FUNCTION_BLOCK FB_HRU EXTENDS FB_CtrlBase
VAR_INPUT
	/// Sensor input
	In_bolHangerDetected: BOOL;
END_VAR
VAR_OUTPUT
	/// Pneumatic cylinder
	Out_bolRotate: BOOL;
	/// Pneumatic cylinder
	Out_bolEject: BOOL;
END_VAR
VAR
	/// Specific interface struct for public access
	SIf: T_Ctrl_SIf_HRU;
	/// Function specific variables
	stSubState: T_Ctrl_Class_StateMachine;
END_VAR
VAR CONSTANT
	///sub States for RELEASE Function
	cSTA_SUB_WAIT_FOR_JOB: INT := 501;
	cSTA_SUB_WAIT_WITH_HANGER: INT := 510;
	cSTA_SUB_ROTATE: INT := 520;
	cSTA_SUB_EJECT: INT := 530;
	cSTA_SUB_RETRACT: INT := 540;
	cSTA_SUB_DONE: INT := 550;
	cSTA_SUB_ERROR: INT := 590;
END_VAR

(*__________________________________________________________________________________________________
¦	
¦	Vistaprint Schweiz GmbH
¦	CH - 8401 Winterthur
¦
¦	www.vistaprint.ch - info@vistaprint.ch
¦___________________________________________________________________________________________________

Function desription:
Hanger rotation unit implementation. 


History:
Version		Date			Author		Comment
---------------------------------------------------------------------------------------------------
0.00.1		25.04.2013		AVME/KVO	Start history
0.00.2		18.09.2013		AVME/MRU	Copied from CYL and renamed to HRU

___________________________________________________________________________________________________*)


IF (me.bolActivate) THEN // cyclic call enabled
	IF (CIf.Info.bolInitDone=FALSE) THEN // first cycle -> init
		CtrlInit();
		CIf.Info.bolInitDone := TRUE;
	ELSE
		CycleStartDuty();
	
		Always();
		
		StateMachine();
		
		CycleEndDuty();
	END_IF
END_IF;

METHOD PROTECTED getCmdState : STRING
VAR_INPUT
	intCmdState: INT;
	bolState: BOOL;
END_VAR
getCmdState := SUPER^.getCmdState(intCmdState:=intCmdState,bolState:=bolState); // get global/base defined cmds/states
IF (getCmdState='') THEN // global not defined get local
	// get string cmd/state string information in runtime
	IF (bolState=FALSE) THEN
		// cmd's
		CASE intCmdState OF
			cCMD_RETRACT: 
				getCmdState := 'cCMD_RETRACT';
			cCMD_EJECT: 
				getCmdState := 'cCMD_EJECT';
			cCMD_ROTATE: 
				getCmdState := 'cCMD_ROTATE';
			cCMD_RUN: 
				getCmdState := 'cCMD_RUN';
		END_CASE;
	ELSE
	
	// states
		CASE intCmdState OF
			cSTA_RETRACTBusy: 
				getCmdState := 'cSTA_RETRACTBusy';
			cSTA_RETRACT: 
				getCmdState := 'cSTA_RETRACT';
			cSTA_EJECTBusy: 
				getCmdState := 'cSTA_EJECTBusy';
			cSTA_EJECT: 
				getCmdState := 'cSTA_EJECT';
			cSTA_ROTATEBusy: 
				getCmdState := 'cSTA_ROTATEBusy';
			cSTA_ROTATE: 
				getCmdState := 'cSTA_ROTATE';
			cSTA_RUNBusy: 
				getCmdState := 'cSTA_RUNBusy';
			cSTA_RUN: 
				getCmdState := 'cSTA_RUN';
				
			// SUB states
			cSTA_SUB_WAIT_FOR_JOB:
				getCmdState := 'cSTA_SUB_WAIT_FOR_JOB';
			cSTA_SUB_WAIT_WITH_HANGER:
				getCmdState := 'cSTA_SUB_WAIT_WITH_HANGER';
			cSTA_SUB_ROTATE:
				getCmdState := 'cSTA_SUB_ROTATE';
			cSTA_SUB_EJECT:
				getCmdState := 'cSTA_SUB_EJECT';
			cSTA_SUB_RETRACT:
				getCmdState := 'cSTA_SUB_RETRACT';
			cSTA_SUB_DONE:
				getCmdState := 'cSTA_SUB_DONE';
			cSTA_SUB_ERROR:
				getCmdState := 'cSTA_SUB_ERROR';

		END_CASE;
	END_IF
END_IF
END_METHOD

METHOD FB_init : BOOL
VAR_INPUT
	///if TRUE, the retain variables are initialized (warm start / cold start)
	bInitRetains: BOOL;
	///if TRUE, the instance afterwards gets moved into the copy code (online change)
	bInCopyCode: BOOL;
END_VAR
VAR
	ii: UINT;
END_VAR
//------------------------------------------------------------------------------------------------------------------------
// to manually change in new FUB implementation!!!
// define valid commands for this controller
FOR ii:= 0 TO (SIZEOF(CIf.Job.aCmdList)/SIZEOF(CIf.Job.aCmdList[0])-1) BY 1 DO
	IF (CIf.Job.aCmdList[ii].intCmd=cCMD_INITIALIZED) THEN
		// found first empty array element
		EXIT;
	END_IF
END_FOR
CIf.Job.aCmdList[ii].intCmd := cCMD_STOP;
CIf.Job.aCmdList[ii].strName := 'Stop'; 
CIf.Job.aCmdList[ii].bolAvailable := TRUE;
ii := ii +1;
CIf.Job.aCmdList[ii].intCmd := cCMD_RETRACT;
CIf.Job.aCmdList[ii].strName := 'Retract';
CIf.Job.aCmdList[ii].bolAvailable := TRUE;
ii := ii +1;
CIf.Job.aCmdList[ii].intCmd := cCMD_EJECT; // for test simulation single answer
CIf.Job.aCmdList[ii].strName := 'EJECT';
CIf.Job.aCmdList[ii].bolAvailable := TRUE;
ii := ii +1;
CIf.Job.aCmdList[ii].intCmd := cCMD_ROTATE; //  MRU 18.09.2013: New command rotate
CIf.Job.aCmdList[ii].strName := 'Rotate'; 
CIf.Job.aCmdList[ii].bolAvailable := TRUE;
ii := ii +1;
CIf.Job.aCmdList[ii].intCmd := cCMD_RUN; // for test simulation single answer
CIf.Job.aCmdList[ii].strName := 'RUN';
CIf.Job.aCmdList[ii].bolAvailable := TRUE;

// set name of class/typ
CIf.Info.strType := 'FB_HRU';

// set alarm class
SIf.Alm[1].eAlmClass := E_AlmClass.TSTOP;
SIf.Alm[1].strText := 'sensor hangerDetected always on'; 
SIf.Alm[2].eAlmClass := E_AlmClass.TSTOP;
SIf.Alm[2].strText := 'sensor hangerDetected always on';
SIf.Alm[3].eAlmClass := E_AlmClass.TSTOP;
SIf.Alm[3].strText := 'sensor hangerDetected always on';
SIf.Alm[4].eAlmClass := E_AlmClass.TSTOP;
SIf.Alm[4].strText := 'Expected Hanger not in Rotation Unit';

//*******************************************************************************
// initial values
//*******************************************************************************

// software configuration
CIf.SwCfg.bolExist := TRUE;
CIf.SwCfg.bolSimulation := FALSE;

// parmeter
SIf.Par.udiEjectTime_ms := 1000;			// No sensor, work with time
SIf.Par.udiRetractTime_ms := 1000;			// No sensor, work with time
SIf.Par.udiRotateTime_ms := 2000;			// No sensor, work with time
SIf.Par.udiWaitForRotate_ms := 4000;		// No sensor, work with time
SIf.Par.udiSimNextHangerTime_ms := 5000;	// For simulation
SIf.Par.udiTimeOutHRU_Hanger_ms := 10000;	// Time out no hanger in rotation unit
END_METHOD

METHOD PROTECTED sta_RETRACTBusy : BOOL
// state implemetation
//--------------------------------------------------------------------------------------
// Entry action
	IF (me.StateMachine.intState<>me.StateMachine.intStateLastCycle) THEN
		me.StateMachine.intStateLastCycle := me.StateMachine.intState;
		
		SIf.Out.bolEject.intern := FALSE;	// Eject Cylinder Valve
		
	END_IF


//--------------------------------------------------------------------------------------
// Cyclic action
	IF (me.StateMachine.intState=me.StateMachine.intStateLastCycle) THEN

		// Simulation
		IF (CIf.SwCfg.bolSimulation) THEN
			;
		END_IF
		
		// State Change Condition
		IF (me.StateMachine.udiTimeInState_ms>SIf.Par.udiRetractTime_ms) THEN
			// Cylinder retracted
			me.StateMachine.intStateNext := cSTA_RETRACT;	
			// timeout extend cylinder 		// Used, if a sensor exist
			// pfbAlarmCtrl^.setAlarm(CIf.Info.intCtrlId,4,0,ADR(SIf.Alm),E_AlmState.RST,CIf.Job.eMe_ActivAlmClass);
			// ELSIF (SIf.In.bolHangerDetected.intern) AND(SIf.In.bolHangerDetected.intern=FALSE) THEN		// Used, if a sensor exist
			// 	me.StateMachine.intStateNext := cSTA_RETRACT;
		ELSIF(me.intCmd=cCMD_STOP) THEN
			me.StateMachine.intStateNext := cSTA_STOPBusy;
		ELSIF(me.intCmd=cCMD_EJECT) THEN
			me.StateMachine.intStateNext := cSTA_EJECTBusy;
		END_IF
	END_IF




//--------------------------------------------------------------------------------------
// Exit action
	IF (me.StateMachine.intState<>me.StateMachine.intStateNext) THEN
		//SIf.Cur.udiMoveTimeRetract := me.StateMachine.udiTimeInState_ms;
		;
	END_IF
END_METHOD

METHOD PROTECTED sta_EJECT : BOOL
// state implemetation
//--------------------------------------------------------------------------------------
// Entry action
	IF (me.StateMachine.intState<>me.StateMachine.intStateLastCycle) THEN
		me.StateMachine.intStateLastCycle := me.StateMachine.intState;

	END_IF


//--------------------------------------------------------------------------------------
// Cyclic action
	IF (me.StateMachine.intState=me.StateMachine.intStateLastCycle) THEN

		// Simulation
		IF (CIf.SwCfg.bolSimulation) THEN
			;
		END_IF
		
		// State Change Condition
		IF (SIf.In.bolHangerDetected.intern) THEN
			// sensor retract always on
			pfbAlarmCtrl^.setAlarm(CIf.Info.intCtrlId,2,0,ADR(SIf.Alm),E_AlmState.RST,CIf.Job.eMe_ActivAlmClass);
			me.StateMachine.intStateNext :=  cSTA_ERROR;
		ELSIF(me.intCmd=cCMD_STOP) THEN
			me.StateMachine.intStateNext := cSTA_STOPBusy;
		ELSIF(me.intCmd=HRU_CmdState.cCMD_RETRACT) THEN
			me.StateMachine.intStateNext := cSTA_RETRACTBusy;
		ELSIF(me.intCmd=HRU_CmdState.cCMD_ROTATE) THEN
			me.StateMachine.intStateNext := cSTA_ROTATEBusy;		
		ELSIF(me.intCmd=cCMD_RUN) THEN
			me.StateMachine.intStateNext := cSTA_RUNBusy;
		END_IF
	END_IF




//--------------------------------------------------------------------------------------
// Exit action
	IF (me.StateMachine.intState<>me.StateMachine.intStateNext) THEN
		;
	END_IF
END_METHOD

METHOD PROTECTED sta_STOP : BOOL
// state implemetation
//--------------------------------------------------------------------------------------
// Entry action
	IF (me.StateMachine.intState<>me.StateMachine.intStateLastCycle) THEN
		me.StateMachine.intStateLastCycle := me.StateMachine.intState;
		
	END_IF


//--------------------------------------------------------------------------------------
// Cyclic action
	IF (me.StateMachine.intState=me.StateMachine.intStateLastCycle) THEN
		
		;
		
		
		// State Change Condition
		IF (me.intCmd=cCMD_OFF) THEN
			// sensor retract always on cylinder
			me.StateMachine.intStateNext :=  cSTA_OFFBusy;
		ELSIF (me.intCmd=cCMD_EJECT) THEN 
			me.StateMachine.intStateNext := cSTA_EJECTBusy;
		ELSIF(me.intCmd=cCMD_RETRACT) THEN
			me.StateMachine.intStateNext := cSTA_RETRACTBusy;
		ELSIF(me.intCmd=cCMD_ROTATE) THEN
			me.StateMachine.intStateNext := cSTA_ROTATEBusy;
		ELSIF (me.intCmd=cCMD_RUN) THEN
			me.StateMachine.intStateNext := cSTA_RUNBusy;
		END_IF
	END_IF




//--------------------------------------------------------------------------------------
// Exit action
	IF (me.StateMachine.intState<>me.StateMachine.intStateNext) THEN
		;
	END_IF
END_METHOD

METHOD PROTECTED sta_RETRACT : BOOL
// state implemetation
//--------------------------------------------------------------------------------------
// Entry action
	IF (me.StateMachine.intState<>me.StateMachine.intStateLastCycle) THEN
		me.StateMachine.intStateLastCycle := me.StateMachine.intState;

	END_IF


//--------------------------------------------------------------------------------------
// Cyclic action
	IF (me.StateMachine.intState=me.StateMachine.intStateLastCycle) THEN

		// Simulation
		IF (CIf.SwCfg.bolSimulation) THEN
			;
		END_IF
		
		// State Change Condition
		IF(me.intCmd=cCMD_STOP) THEN
			me.StateMachine.intStateNext := cSTA_STOPBusy;
		ELSIF(me.intCmd=HRU_CmdState.cCMD_EJECT) THEN
			me.StateMachine.intStateNext := cSTA_EJECTBusy;
		ELSIF(me.intCmd=HRU_CmdState.cCMD_ROTATE) THEN
			me.StateMachine.intStateNext := cSTA_ROTATEBusy;
		ELSIF(me.intCmd=cCMD_RUN) THEN
			me.StateMachine.intStateNext := cSTA_RUNBusy;
		END_IF
	END_IF




//--------------------------------------------------------------------------------------
// Exit action
	IF (me.StateMachine.intState<>me.StateMachine.intStateNext) THEN
		;
	END_IF
END_METHOD

METHOD PROTECTED sta_RUNBusy : BOOL
// state implemetation
//--------------------------------------------------------------------------------------
// Entry action
	IF (me.StateMachine.intState<>me.StateMachine.intStateLastCycle) THEN
		me.StateMachine.intStateLastCycle := me.StateMachine.intState;

		me.SubStateMachine.intState := cSTA_SUB_WAIT_FOR_JOB; 		// init sub state machine
		me.SubStateMachine.intStateNext := cSTA_SUB_WAIT_FOR_JOB; 	// init sub state machine
		
		fbSimulationTimer.IN := FALSE;
		fbSimulationTimer.PT := UDINT_TO_TIME(SIf.Par.udiSimNextHangerTime_ms);
		fbSimulationTimer(); // set time/reset timer
		//fbSimulationTimer.IN := TRUE; // start timer
	END_IF


//--------------------------------------------------------------------------------------
// Cyclic action
	IF (me.StateMachine.intState=me.StateMachine.intStateLastCycle) THEN

		// Simulation
		IF (CIf.SwCfg.bolSimulation) THEN
			fbSimulationTimer(); // simulation time
		END_IF

		//--------------------------------------------------------------------------------------
		// sub state machine for sequence
		CASE me.SubStateMachine.intState OF
			cSTA_SUB_WAIT_FOR_JOB:
				IF (me.SubStateMachine.intState<>me.SubStateMachine.intStateLastCycle) THEN
					me.SubStateMachine.intStateLastCycle := me.SubStateMachine.intState;
				END_IF
				
				// Simulation
				IF (CIf.SwCfg.bolSimulation AND NOT SIf.In.bolHangerDetected.intern) THEN
					fbSimulationTimer.IN := TRUE; // start timer
				END_IF
				IF (fbSimulationTimer.Q) THEN
					SIf.In.bolHangerDetected.intern := TRUE; 	// Hanger in HRU
					fbSimulationTimer.IN := FALSE; 				// Stop timer
				END_IF
				
				// State Change Condition
				// Check error if possible
				IF (SIf.In.bolHangerDetected.intern) THEN
					me.SubStateMachine.intStateNext := cSTA_SUB_WAIT_WITH_HANGER;
				END_IF
				
				// Time out expected hanger is not arrived
				IF (me.SubStateMachine.udiTimeInState_ms > SIf.Par.udiTimeOutHRU_Hanger_ms) THEN	// Hanger Rotation Unit time out waiting
					pfbAlarmCtrl^.setAlarm(CIf.Info.intCtrlId,4,0,ADR(SIf.Alm),E_AlmState.RST,CIf.Job.eMe_ActivAlmClass);
					me.SubStateMachine.intStateNext := cSTA_SUB_ERROR;
				END_IF
		//--------------------------------------------------------------------------------------
			cSTA_SUB_WAIT_WITH_HANGER:
				IF (me.SubStateMachine.intState<>me.SubStateMachine.intStateLastCycle) THEN
					me.SubStateMachine.intStateLastCycle := me.SubStateMachine.intState;
				END_IF
				
				// State Change Condition
				// Check error if possible
				IF (me.SubStateMachine.udiTimeInState_ms >= SIf.Par.udiWaitForRotate_ms) THEN
					me.SubStateMachine.intStateNext := cSTA_SUB_ROTATE;
				END_IF
		//--------------------------------------------------------------------------------------
			cSTA_SUB_ROTATE:
				IF (me.SubStateMachine.intState<>me.SubStateMachine.intStateLastCycle) THEN
					me.SubStateMachine.intStateLastCycle := me.SubStateMachine.intState;
					SIf.Out.bolRotate.intern := NOT SIf.Out.bolRotate.intern;	// Rotate in other direction
				END_IF
				
				
				// State Change Condition
				// Check error if possible
				IF (me.SubStateMachine.udiTimeInState_ms >= SIf.Par.udiRotateTime_ms) THEN
					me.SubStateMachine.intStateNext := cSTA_SUB_EJECT;
				END_IF
		//--------------------------------------------------------------------------------------
			cSTA_SUB_EJECT:
				IF (me.SubStateMachine.intState<>me.SubStateMachine.intStateLastCycle) THEN
					me.SubStateMachine.intStateLastCycle := me.SubStateMachine.intState;
				END_IF
				
				SIf.Out.bolEject.intern := TRUE;	// Eject Cylinder Valve
				
				// Simulation
				IF (CIf.SwCfg.bolSimulation) THEN
					SIf.In.bolHangerDetected.intern := FALSE; // Hanger is leaving the HRU
				END_IF
				
				// State Change Condition
				// Check error if possible
				IF (me.SubStateMachine.udiTimeInState_ms > SIf.Par.udiEjectTime_ms) THEN
					IF (SIf.In.bolHangerDetected.intern) THEN
					// sensor Hanger detected always on
						pfbAlarmCtrl^.setAlarm(CIf.Info.intCtrlId,3,0,ADR(SIf.Alm),E_AlmState.RST,CIf.Job.eMe_ActivAlmClass);
						me.SubStateMachine.intStateNext := cSTA_SUB_ERROR;
					ELSE
						// Hanger ejected
						me.SubStateMachine.intStateNext := cSTA_SUB_RETRACT;
					END_IF
				END_IF
		//--------------------------------------------------------------------------------------
			cSTA_SUB_RETRACT:
				IF (me.SubStateMachine.intState<>me.SubStateMachine.intStateLastCycle) THEN
					me.SubStateMachine.intStateLastCycle := me.SubStateMachine.intState;
				END_IF
				
				SIf.Out.bolEject.intern := FALSE;	// Eject Cylinder Valve

				// State Change Condition
				// Check error if possible
				IF (me.SubStateMachine.udiTimeInState_ms >= SIf.Par.udiRetractTime_ms) THEN
					me.SubStateMachine.intStateNext := cSTA_SUB_DONE;
				END_IF
		//--------------------------------------------------------------------------------------
			cSTA_SUB_DONE:
				//CIf.Job.intACmd:=cSTA_DONE; 	// Not necessary
				;								// do nothing, just for state change
		//--------------------------------------------------------------------------------------
			cSTA_SUB_ERROR:
				IF (me.SubStateMachine.intState<>me.SubStateMachine.intStateLastCycle) THEN
					me.SubStateMachine.intStateLastCycle := me.SubStateMachine.intState;
				END_IF
				
				SIf.Out.bolEject.intern := FALSE;	// Eject Cylinder Valve
				
				// State Change Condition
				// No change, going over an other main state
		//--------------------------------------------------------------------------------------
		END_CASE
		
		// Do in every cycle
		CIf.Job.strSubState := THIS^.getCmdState(intCmdState:=me.SubStateMachine.intState,bolState:=TRUE);
		IF (me.SubStateMachine.intState<>me.SubStateMachine.intStateNext) THEN
			me.SubStateMachine.intState := me.SubStateMachine.intStateNext;  // set next state for next cycle
			me.SubStateMachine.udiTimeInState_ms := 0; // reset timer
			// log state change -> open point
		ELSE
			// increment time in state	
			me.SubStateMachine.udiTimeInState_ms := me.SubStateMachine.udiTimeInState_ms + me.FUBInfo.udiSample_ms;
		END_IF
		
				
		// State Change Condition	
		IF me.SubStateMachine.intState = cSTA_SUB_ERROR THEN
			me.StateMachine.intStateNext :=  cSTA_ERROR;
		ELSIF(me.SubStateMachine.intState = cSTA_SUB_DONE) THEN
			me.StateMachine.intStateNext := cSTA_RUN;
		ELSIF((me.SubStateMachine.intState = cSTA_SUB_WAIT_FOR_JOB) AND(me.intCmd=cCMD_STOP)) THEN
			me.StateMachine.intStateNext := cSTA_STOPBusy;
		//ELSIF((me.SubStateMachine.intState = cSTA_SUB_WAIT_FOR_JOB) AND(me.intCmd=cCMD_OFF)) THEN // Done by BaseCtrl.Always
		//	me.StateMachine.intStateNext := cSTA_OFFBusy;
		END_IF
	END_IF


//--------------------------------------------------------------------------------------
// Exit action
	IF (me.StateMachine.intState<>me.StateMachine.intStateNext) THEN
		;
	END_IF
END_METHOD

METHOD PROTECTED sta_RUN : BOOL
// state implemetation
//--------------------------------------------------------------------------------------
// Entry action
	IF (me.StateMachine.intState<>me.StateMachine.intStateLastCycle) THEN
		me.StateMachine.intStateLastCycle := me.StateMachine.intState;
				
	END_IF


//--------------------------------------------------------------------------------------
// Cyclic action
	IF (me.StateMachine.intState=me.StateMachine.intStateLastCycle) THEN

		// Simulation
		IF (CIf.SwCfg.bolSimulation) THEN
			;
		END_IF
		
		// Cyclicle action
		
		
		// State Change Condition
		IF (TRUE) THEN		// Stop after every cycle -> cSTA_DONE
			me.StateMachine.intStateNext := cSTA_STOPBusy;
		ELSIF (me.intCmd=cCMD_STOP) THEN
			me.StateMachine.intStateNext :=  cSTA_STOPBusy;	
		END_IF
	END_IF


//--------------------------------------------------------------------------------------
// Exit action
	IF (me.StateMachine.intState<>me.StateMachine.intStateNext) THEN
		;
	END_IF
END_METHOD

METHOD getCtrlSIf : POINTER TO T_Ctrl_SIf_HRU
getCtrlSIf := ADR(SIf);
END_METHOD

METHOD PROTECTED sta_ROTATEBusy : BOOL
// state implemetation
//--------------------------------------------------------------------------------------
// Entry action
	IF (me.StateMachine.intState<>me.StateMachine.intStateLastCycle) THEN
		me.StateMachine.intStateLastCycle := me.StateMachine.intState;
		
		SIf.Out.bolRotate.intern := NOT SIf.Out.bolRotate.intern;	// Rotate in other direction
		
	END_IF


//--------------------------------------------------------------------------------------
// Cyclic action
	IF (me.StateMachine.intState=me.StateMachine.intStateLastCycle) THEN

		// Simulation
		IF (CIf.SwCfg.bolSimulation) THEN
			;
		END_IF
		
		// State Change Condition
		IF (me.StateMachine.udiTimeInState_ms>SIf.Par.udiRotateTime_ms) THEN
			me.StateMachine.intStateNext :=  cSTA_ROTATE;
		ELSIF(me.intCmd=cCMD_OFF) THEN
			me.StateMachine.intStateNext := cSTA_OFFBusy;
		ELSIF(me.intCmd=cCMD_STOP) THEN
			me.StateMachine.intStateNext := cSTA_STOPBusy;
		END_IF
	END_IF




//--------------------------------------------------------------------------------------
// Exit action
	IF (me.StateMachine.intState<>me.StateMachine.intStateNext) THEN
		//SIf.Cur.udiMoveTimeRetract := me.StateMachine.udiTimeInState_ms;
		;
	END_IF
END_METHOD

METHOD PROTECTED sta_STOPBusy : BOOL
// state implemetation
//--------------------------------------------------------------------------------------
// Entry action
	IF (me.StateMachine.intState<>me.StateMachine.intStateLastCycle) THEN
		me.StateMachine.intStateLastCycle := me.StateMachine.intState;
		
	END_IF


//--------------------------------------------------------------------------------------
// Cyclic action
	IF (me.StateMachine.intState=me.StateMachine.intStateLastCycle) THEN
		
		// switch off?
		// SIf.Out.bolEject.intern := FALSE;	// Eject Cylinder Valve
		
		// State Change Condition
		IF (FALSE) THEN
			;
		ELSIF (TRUE) THEN
			me.StateMachine.intStateNext := cSTA_STOP;
		END_IF
	END_IF




//--------------------------------------------------------------------------------------
// Exit action
	IF (me.StateMachine.intState<>me.StateMachine.intStateNext) THEN
		;
	END_IF
END_METHOD

METHOD PROTECTED sta_OFF : BOOL
// state implemetation
//--------------------------------------------------------------------------------------
// Entry action
	IF (me.StateMachine.intState<>me.StateMachine.intStateLastCycle) THEN
		me.StateMachine.intStateLastCycle := me.StateMachine.intState;
		
	END_IF


//--------------------------------------------------------------------------------------
// Cyclic action
	IF (me.StateMachine.intState=me.StateMachine.intStateLastCycle) THEN
		
		;
		
		
		// State Change Condition
		IF (me.intCmd=cCMD_STOP) THEN
			me.StateMachine.intStateNext :=  cSTA_STOPBusy;
		ELSIF (me.intCmd=HRU_CmdState.cCMD_EJECT) THEN 
			me.StateMachine.intStateNext := cSTA_EJECTBusy;
		ELSIF(me.intCmd=HRU_CmdState.cCMD_RETRACT) THEN
			me.StateMachine.intStateNext := cSTA_RETRACTBusy;
		ELSIF(me.intCmd=HRU_CmdState.cCMD_ROTATE) THEN
			me.StateMachine.intStateNext := cSTA_ROTATEBusy;
		ELSIF(me.intCmd=cCMD_RUN) THEN
			me.StateMachine.intStateNext := cSTA_RUNBusy;
		END_IF
	END_IF




//--------------------------------------------------------------------------------------
// Exit action
	IF (me.StateMachine.intState<>me.StateMachine.intStateNext) THEN
		;
	END_IF
END_METHOD

METHOD PROTECTED sta_OFFBusy : BOOL
// state implemetation
//--------------------------------------------------------------------------------------
// Entry action
	IF (me.StateMachine.intState<>me.StateMachine.intStateLastCycle) THEN
		me.StateMachine.intStateLastCycle := me.StateMachine.intState;
		
	END_IF


//--------------------------------------------------------------------------------------
// Cyclic action
	IF (me.StateMachine.intState=me.StateMachine.intStateLastCycle) THEN
		
		// switch off?
		// SIf.Out.bolEject.intern := FALSE;	// Eject Cylinder Valve
		
		// State Change Condition
		IF (FALSE) THEN
			;
		ELSIF (TRUE) THEN
			me.StateMachine.intStateNext := cSTA_OFF;
		END_IF
	END_IF




//--------------------------------------------------------------------------------------
// Exit action
	IF (me.StateMachine.intState<>me.StateMachine.intStateNext) THEN
		;
	END_IF
END_METHOD

METHOD PROTECTED IoOutBridge : BOOL
// digitale and analoge inputs read from hardware or forcing
IF (CIf.SwCfg.bolSimulation = FALSE) THEN
	setOutBol(CIf.Job.bolIoForce ,ADR(SIf.Out.bolEject));
	setOutBol(CIf.Job.bolIoForce ,ADR(SIf.Out.bolRotate));
	
	THIS^.Out_bolEject := SIf.Out.bolEject.map;
	THIS^.Out_bolRotate := SIf.Out.bolRotate.map;
END_IF
END_METHOD

METHOD PROTECTED StateMachine : BOOL
SUPER^.StateMachine();

// main statemachine of base controller
CASE me.StateMachine.intState OF
	cSTA_ROTATEBusy: 
        THIS^.sta_ROTATEBusy();
    cSTA_ROTATE: 
        THIS^.sta_ROTATE();
	cSTA_RETRACTBusy: 
        THIS^.sta_RETRACTBusy();
    cSTA_RETRACT: 
        THIS^.sta_RETRACT();
    cSTA_EJECTBusy:				// Eject 
        THIS^.sta_EJECTBusy();
    cSTA_EJECT: 
        THIS^.sta_EJECT();
	cSTA_RUNBusy: 
        THIS^.sta_RUNBusy();	// Auto (Wait - Rotate - Eject - Retract)
    cSTA_RUN: 
        THIS^.sta_RUN();
	cSTA_STOPBusy: 				// Rotate rests in his Position, Ejector in Retract Position
        THIS^.sta_STOPBusy();
    cSTA_STOP: 
        THIS^.sta_STOP();
		
END_CASE;
END_METHOD

METHOD PROTECTED sta_EJECTBusy : BOOL
// state implemetation
//--------------------------------------------------------------------------------------
// Entry action
	IF (me.StateMachine.intState<>me.StateMachine.intStateLastCycle) THEN
		me.StateMachine.intStateLastCycle := me.StateMachine.intState;

	END_IF


//--------------------------------------------------------------------------------------
// Cyclic action
	IF (me.StateMachine.intState=me.StateMachine.intStateLastCycle) THEN

		// Simulation
		IF (CIf.SwCfg.bolSimulation) THEN
			;
		END_IF
		
		//no change action
		SIf.Out.bolEject.intern := TRUE;	// Eject Cylinder Valve
		
		
		// State Change Condition
		IF (me.StateMachine.udiTimeInState_ms>SIf.Par.udiEjectTime_ms) THEN
			IF (SIf.In.bolHangerDetected.intern) THEN
				// sensor Hanger detected always on
				pfbAlarmCtrl^.setAlarm(CIf.Info.intCtrlId,1,0,ADR(SIf.Alm),E_AlmState.RST,CIf.Job.eMe_ActivAlmClass);
				me.StateMachine.intStateNext :=  cSTA_ERROR;
			ELSE
				// Hanger ejected
				me.StateMachine.intStateNext := cSTA_EJECT;	
			END_IF
		ELSIF(me.intCmd=cCMD_STOP) THEN
			me.StateMachine.intStateNext := cSTA_STOPBusy;
		ELSIF(me.intCmd=HRU_CmdState.cCMD_RETRACT) THEN
			me.StateMachine.intStateNext := cSTA_RETRACTBusy;
		END_IF
	END_IF




//--------------------------------------------------------------------------------------
// Exit action
	IF (me.StateMachine.intState<>me.StateMachine.intStateNext) THEN
		;
	END_IF
END_METHOD

METHOD PROTECTED IoInBridge : BOOL
// digitale and analoge inputs read from hardware or forcing
SIf.In.bolHangerDetected .map := THIS^.In_bolHangerDetected;

IF (CIf.SwCfg.bolSimulation = FALSE) THEN
	getInBol(CIf.Job.bolIoForce,ADR(SIf.In.bolHangerDetected));
ELSE
	//simulation of global IO
END_IF
END_METHOD

METHOD PROTECTED Always : BOOL
SUPER^.Always();

IF (me.StateMachine.intState<>cSTA_SINGLE_ANSWER) THEN
	;
END_IF


// Always change actions in Base Library
// ----------------------------------------------------------------------------------
// overrule error always from base -> no EOFF State!! in EOFF go to OFF
IF (me.StateMachine.intStateNext = cSTA_EOFFBusy) THEN
	IF (me.StateMachine.intState=cSTA_OFF) THEN
		me.StateMachine.intStateNext := cSTA_OFF;
	ELSE // stay in OFF
		me.StateMachine.intStateNext := cSTA_OFFBusy;
	END_IF
END_IF
END_METHOD

METHOD PROTECTED sta_ROTATE : BOOL
// state implemetation
//--------------------------------------------------------------------------------------
// Entry action
	IF (me.StateMachine.intState<>me.StateMachine.intStateLastCycle) THEN
		me.StateMachine.intStateLastCycle := me.StateMachine.intState;

	END_IF


//--------------------------------------------------------------------------------------
// Cyclic action
	IF (me.StateMachine.intState=me.StateMachine.intStateLastCycle) THEN

		// Simulation
		IF (CIf.SwCfg.bolSimulation) THEN
			;
		END_IF
		
		
		IF(me.intCmd=cCMD_OFF) THEN
			me.StateMachine.intStateNext := cSTA_OFFBusy;
		ELSIF(me.intCmd=cCMD_STOP) THEN
			me.StateMachine.intStateNext := cSTA_STOPBusy;
		ELSIF(me.intCmd=HRU_CmdState.cCMD_EJECT) THEN
			me.StateMachine.intStateNext := cSTA_EJECTBusy;
		ELSIF(me.intCmd=HRU_CmdState.cCMD_RETRACT) THEN
			me.StateMachine.intStateNext := cSTA_RETRACTBusy;
		ELSIF(me.intCmd=cCMD_RUN) THEN
			me.StateMachine.intStateNext := cSTA_RUNBusy;
		END_IF
	END_IF




//--------------------------------------------------------------------------------------
// Exit action
	IF (me.StateMachine.intState<>me.StateMachine.intStateNext) THEN
		;
	END_IF
END_METHOD

END_FUNCTION_BLOCK

(* stored: Version 1.1.0.1, ProductVersion 3.1.0.19
   POU FB_HRU: Id {e7da98a9-648f-45a2-b6cd-3c8fb8ea4a27}
   Method getCmdState: Id {f92c1110-dbbf-41b3-98a4-d1e3072092cf}
   Method FB_init: Id {d643d3ce-c3a3-4949-99ff-f9349508240f}
   Method sta_RETRACTBusy: Id {320f6078-e245-4d47-a49f-217085321fcb}
   Method sta_EJECT: Id {14a531a2-46cf-4064-847e-c670d34b589f}
   Method sta_STOP: Id {6858f917-2fab-4582-a04f-9a9509e1f096}
   Method sta_RETRACT: Id {d8ab7be5-af2e-45de-a83b-eaced7a8b732}
   Method sta_RUNBusy: Id {4fa02b40-e25e-4f78-9cb6-d34028e86296}
   Method sta_RUN: Id {452e79f6-9c6d-4c20-b538-1c5573f25e88}
   Method getCtrlSIf: Id {1b617f7b-a794-4338-92da-3e6a3f0e465f}
   Method sta_ROTATEBusy: Id {29398fc9-21df-48af-abd1-bb4882462baf}
   Method sta_STOPBusy: Id {9faad390-abfc-46ee-b257-7bb0c5b9e8fe}
   Method sta_OFF: Id {be156e11-04eb-4142-8c99-c662a9103b70}
   Method sta_OFFBusy: Id {66438238-6d7d-4718-a8ce-677a732faa2d}
   Method IoOutBridge: Id {1a8b54f3-45d9-4433-8efa-9df953e7be19}
   Method StateMachine: Id {5c20de26-01e9-4464-bd05-2f21273be419}
   Method sta_EJECTBusy: Id {4877cc40-a1b7-4684-af1e-67b223137e67}
   Method IoInBridge: Id {593af27c-1a76-48d5-b3a4-1932fa43020d}
   Method Always: Id {107a1b23-5daf-4da3-b36f-d0e0914536ad}
   Method sta_ROTATE: Id {ae137dec-2217-4c39-8664-d4bc46bfb94a} *)
